(*
Generates TIME in 100ns since 1ST January 1970.
Bases on Tc2_System.F_GetSystemTime FUNCTION.
The result can be adjusted through the nOffset variable.
*)
FUNCTION GetUnixTime : ULINT
VAR_INPUT
	nOffset : LINT := 0;
END_VAR
VAR
END_VAR

GetUnixTime := Tc2_System.F_GetSystemTime() - LINT_TO_ULINT(11_644_473_678_000_000_0 + nOffset);

END_FUNCTION

(* stored: Version 1.1.0.1
   POU GetUnixTime: Id {9256dbe0-970c-46b2-beb0-50dc80b906e9}, SpecialFunc None *)
